{attribute 'GeneratedUsingTerminal: EK1100-0000-0018'}
{attribute addProperty BoxType "EK1100-0000-0018"}
{attribute addProperty Id "Beckhoff_EJ9xxxEK1122Beckhoff_EJ9xxxEK1122_C80E1DB32A_0001_EJ9001_0000_0016EJ9001_1FC0878B2A_0002_EJ9505_0000_0016EJ9505_19A4723D6A_0003_EJ9576_0000_0018EJ9576_04A95C1A20A_0004_EJ9576_0000_0019EJ9576_E580EC2021A_0005_EJ9576_0000_0020EJ9576_AF0E5C2A20A_0006_EJ9576_0000_0022EJ9576_F397F1AC21"}
{attribute addProperty CRC "2549571589"}
{attribute addProperty Size "92"}
TYPE Beckhoff_EJ9xxx_97F76005 EXTENDS EK1100_1FC0878B :
STRUCT
	{attribute addProperty Name "Beckhoff_EJ9xxxEK1122"}
	{attribute addProperty PreviousPort "Beckhoff EJ9xxx : B"}
	Beckhoff_EJ9xxxEK1122 : Beckhoff_EJ9xxxEK1122_C80E1DB3;
	{attribute addProperty Name "A_0001_EJ9001_0000_0016"}
	{attribute addProperty PreviousPort "Beckhoff EJ9xxxEK1122 : C"}
	A_0001_EJ9001_0000_0016 : EJ9001_1FC0878B;
	{attribute addProperty Name "A_0002_EJ9505_0000_0016"}
	{attribute addProperty PreviousPort "A_0001(EJ9001-0000-0016) : B"}
	A_0002_EJ9505_0000_0016 : EJ9505_19A4723D;
	{attribute addProperty Name "A_0003_EJ9576_0000_0018"}
	{attribute addProperty PreviousPort "A_0002(EJ9505-0000-0016) : B"}
	A_0003_EJ9576_0000_0018 : EJ9576_04A95C1A;
	{attribute addProperty Name "A_0004_EJ9576_0000_0019"}
	{attribute addProperty PreviousPort "A_0003(EJ9576-0000-0018) : B"}
	A_0004_EJ9576_0000_0019 : EJ9576_E580EC20;
	{attribute addProperty Name "A_0005_EJ9576_0000_0020"}
	{attribute addProperty PreviousPort "A_0004(EJ9576-0000-0019) : B"}
	A_0005_EJ9576_0000_0020 : EJ9576_AF0E5C2A;
	{attribute addProperty Name "A_0006_EJ9576_0000_0022"}
	{attribute addProperty PreviousPort "A_0005(EJ9576-0000-0020) : B"}
	A_0006_EJ9576_0000_0022 : EJ9576_F397F1AC;
END_STRUCT
END_TYPE

(* stored: Version 1.2.0.0, ProductVersion 3.1.4024.9
   DUT Beckhoff_EJ9xxx_97F76005: Id {c125de06-645a-4896-8249-1b0d6e85dca2} *)
